ABB RAPID module: A083_DataTask_Rob.mod

MODULE A083_DataTask_Rob
    !***********************************************************************************
    !
    ! ETH Zurich / NCCR Digital Fabrication
    ! HIB C51 / Stefano-Franscini-Platz 1
    ! CH-8093 Zurich
    !
    !***********************************************************************************
    !
    ! PROJECT     :  A083 Augmented-Timber
    !
    ! FUNCTION    :  Includ all Task Data's for Project
    !
    ! AUTHOR      :  Philippe Fleischmann
    !
    ! EMAIL       :  fleischmann@arch.ethz.ch
    !
    ! HISTORY     :  2022.01.20
    !
    ! Copyright   :  ETH Zurich (CH) 2022
    !
    !***********************************************************************************

    !************************************************
    ! Declaration :     bool
    !************************************************
    !
    TASK PERS bool b_A083_MyBool:=FALSE;

    !************************************************
    ! Declaration :     num
    !************************************************
    !
    TASK PERS num n_A083_MyNum:=0;

    !************************************************
    ! Declaration :     string
    !************************************************
    !
    TASK PERS string st_A083_MyString:="";

    !************************************************
    ! Declaration :     tooldata
    !************************************************
    !
    TASK PERS tooldata t_A083_MyTool:=[TRUE,[[0,0,0],[1,0,0,0]],[0,[0,0,0],[1,0,0,0],0,0,0]];
    TASK PERS tooldata t_A083_RefTip:=[TRUE,[[0,0,250],[1,0,0,0]],[2,[0,0,50],[1,0,0,0],0,0,0]];

    !************************************************
    ! Declaration :     wobjdata
    !************************************************
    !
    TASK PERS wobjdata ob_A083_MyWobjdata:=[FALSE,TRUE,"",[[0,0,0],[1,0,0,0]],[[0,0,0],[1,0,0,0]]];
    TASK PERS wobjdata ob_A083_Wobj_Place:=[FALSE,TRUE,"",[[-207.311,-1071,-39.4772],[0.575754,0.000199967,0.000151784,-0.817623]],[[0,0,0],[1,0,0,0]]];
    TASK PERS wobjdata ob_A083_Wobj_Pick:=[FALSE,TRUE,"",[[-1049.15,-568.768,-42.1385],[0.233655,-0.00369194,0.000702063,0.972312]],[[0,0,0],[1,0,0,0]]];

    !************************************************
    ! Declaration :     jointtarget
    !************************************************
    !
    TASK PERS jointtarget jp_A083_MyJointtarget:=[[0,0,0,0,0,0],[9E9,9E9,9E9,9E9,9E9,9E9]];

    !************************************************
    ! Declaration :     robtarget
    !************************************************
    !
    TASK PERS robtarget p_A083_MyRobtarget:=[[0,0,0],[1,0,0,0],[0,0,0,0],[9E9,9E9,9E9,9E9,9E9,9E9]];
    !
    ! Demo points
    TASK PERS robtarget p_A083_Home:=[[0,0,300],[0.247354,0.8325,-0.437708,0.232748],[-2,1,-3,1],[-301.6,9E+09,9E+09,9E+09,9E+09,9E+09]];
    TASK PERS robtarget p_A083_Pick:=[[18,31,1],[0.247354,0.8325,-0.437708,0.232748],[-2,1,-3,1],[-301.6,9E+09,9E+09,9E+09,9E+09,9E+09]];

    !************************************************
    ! Declaration :     speeddata
    !************************************************
    !
    TASK PERS speeddata v_A083_MySpeed:=[0,0,0,0];
ENDMODULE
